FUNCTION_BLOCK FB_Movement_Gcode
VAR_INPUT
	bExecute : BOOL;
END_VAR
VAR_OUTPUT
	bBusy : BOOL;
	bError : BOOL;
	bFinished : BOOL;
	initial : R_TRIG;
END_VAR
VAR
	gcodeagent : FB_GcodeAgent;
	// define kinematics objects
	fbMover : FB_HbotMovement;
	fbHome : FB_HbotHome;
	sGodeFileName : STRING;
	caseswitch : (init, prep, movement, end, error);
END_VAR

initial(CLK := bExecute);
IF initial.Q THEN // on initial trigger, run initilsation case to initiate gcode and reset variables
	caseswitch := init;
	bFinished := FALSE;
	bBusy := TRUE;
	gcodeagent.bEnd := FALSE;
END_IF
CASE caseswitch OF
	init:
		IF sGodeFileName <> '' THEN
			IF bExecute AND NOT bError THEN
			gcodeagent(sGcodeFile := sGodeFileName, sFBName := 'MovementTypeSelector.fbGcode.gcodeagent', bExecute := bExecute);
			// run gcode agent python script
			IF NOT gcodeagent.Process.BUSY THEN 
				caseswitch := prep;
			END_IF
		END_IF
		END_IF
	prep:
		fbMover( bExecute := FALSE, StepperA := GVL.StepperReferenceA, StepperB := GVL.StepperReferenceB); // stop all movement
		IF gcodeagent.bWriteDone THEN // wait for gcode agent to write a new line before going to next step
			caseswitch := movement;
		END_IF
		IF gcodeagent.bEnd THEN
			caseswitch := end; // if gcode agent sends a end command, go to end case
		END_IF
	movement:
		fbMover(MovementMode := fbMover.MoveAbsolute,
				rLinearSpeed := 60,
				rCurrentX := HbotForwardKinematics.rCurrentX,
				rCurrentY := HbotForwardKinematics.rCurrentY,
				rDeltaX := gcodeagent.x,
				rDeltaY := gcodeagent.y,
				bExecute := TRUE,
				StepperA := GVL.StepperReferenceA,
				StepperB := GVL.StepperReferenceB); // once gcode is received, move to positions
				 
		IF fbMover.bError THEN
			caseswitch := error; //catch errors
		ELSIF fbMover.bDone THEN
			caseswitch := prep; // if it is done, go to the prep switch case
			gcodeagent.bNextLine := TRUE; // send signal to python script to show that the movement is completed
		END_IF
	end:
		bFinished := TRUE;
		bBusy := FALSE;
		gcodeagent(sGcodeFile := 'choppt.gcode', sFBName := 'MovementTypeSelector.fbGcode.gcodeagent', bExecute := FALSE);
	error:
		bError := TRUE;
END_CASE

END_FUNCTION_BLOCK

(* stored: Version 1.1.0.1, ProductVersion 3.1.4024.11
   POU FB_Movement_Gcode: Id {5782bb99-49b0-437e-b251-04e1fb995da8}, SpecialFunc None *)
